// TIA Portal project "Asansör" (V16)

(* hardware
DEVICE "HMI_1"  TP900 Comfort
   slot 0: "HMI_1"  TP900 Comfort  6AV2 124-0JC01-0AX0  16.0.0.0
   slot 1: "HMI_RT_1"  TP900 Comfort  6AV2 124-0JC01-0AX0  16.0.0.0
   slot 5: "HMI_1.IE_CP_1"  PROFINET Interface  16.0.0.0
      slot 1: "PROFINET Interface_1"  PROFINET Interface
         slot 1: "Port_1"  Port
         slot 2: "Port_2"  Port
   slot 7: "HMI_1.MPI/DP_CP_1"  MPI/DP Interface  16.0.0.0
DEVICE "S71500/ET200MP station_1"  S7-1500 station
   slot 0: "Rail_0"  Rack  6ES7 590-1***0-0AA0
   slot 1: "PLC_1"  CPU 1513-1 PN  6ES7 513-1AL00-0AB0  V1.8
      slot 3: "CPU display_1"  6ES7591-1AA00-0AA0
      slot 32768: "PROFINET interface_1"  X1
         slot 32769: "Port_1"  X1 P1
         slot 32770: "Port_2"  X1 P2
*)

// ===== PLC "PLC_1"  CPU 1513-1 PN =====

VAR_GLOBAL   // PLC tag table "Default tag table"
   "Start" AT %M0.0 : Bool;
   "Start-System" AT %M0.1 : Bool;
   "P_TRIG" AT %M5.0 : Bool;
   "Stop" AT %M0.2 : Bool;
   "Low_Sensor" AT %M0.3 : Bool;
   "High_Sensor" AT %M0.4 : Bool;
   "P_TRIG1" AT %M5.1 : Bool;
   "Floor 1 button" AT %M0.5 : Bool;
   "P_TRIG2" AT %M5.2 : Bool;
   "Floor 1_Memory" AT %M0.6 : Bool;
   "Floor1_Sensor" AT %M0.7 : Bool;
   "P_TRIG3" AT %M5.3 : Bool;
   "Floor 2 button" AT %M1.0 : Bool;
   "P_TRIG4" AT %M5.4 : Bool;
   "Floor 2_Memory" AT %M1.1 : Bool;
   "Floor2_Sensor" AT %M1.2 : Bool;
   "P_TRIG5" AT %M5.5 : Bool;
   "Floor 3 button" AT %M1.3 : Bool;
   "Floor 3_Memory" AT %M1.4 : Bool;
   "P_TRIG6" AT %M5.6 : Bool;
   "Floor3_Sensor" AT %M1.5 : Bool;
   "P_TRIG7" AT %M5.7 : Bool;
   "P_TRIG8" AT %M6.1 : Bool;
   "Motor_Memory" AT %M1.6 : Bool;
   "Motor_Up" AT %M1.7 : Bool;
   "P_TRIG9" AT %M6.2 : Bool;
   "Memory2" AT %M2.0 : Bool;
   "Memory3" AT %M2.1 : Bool;
   "P_TRIG10" AT %M6.3 : Bool;
   "Motor_asagımemory" AT %M2.2 : Bool;
   "Motor_Down" AT %M2.3 : Bool;
   "P_TRIG11" AT %M6.4 : Bool;
   "Memory4" AT %M2.4 : Bool;
   "Memory5" AT %M2.5 : Bool;
END_VAR

DATA_BLOCK "Elevator"   // DB1
{ S7_Optimized_Access := 'TRUE' }
VERSION : 0.1
   VAR
      "Start System" : Bool;
      "Start--Stop" : Bool;
      "0_Floor" : Bool;
      "1_Floor" : Bool;
      "2_Floor" : Bool;
      Fan : Bool;
      Low_Sensor : Bool;
      High_Sensor : Bool;
      "1_Floor_Button" : Bool;
      "1_Floor_Sensor" : Bool;
      "2_Floor_Button" : Bool;
      "2_Floor_Sensor" : Bool;
      "3_Floor_Button" : Bool;
      "3_Floor_Sensor" : Bool;
      Motor_Up : Bool;
   END_VAR
BEGIN
END_DATA_BLOCK

ORGANIZATION_BLOCK "Main"   // OB1, LAD, ProgramCycle
TITLE = "Main Program Sweep (Cycle)"
{ S7_Optimized_Access := 'TRUE' }
VERSION : 0.1
   VAR_INPUT
      Initial_Call : Bool;   // Initial call of this OB
      Remanence : Bool;   // =True, if remanent data are available
   END_VAR
   VAR_TEMP   // added for the SCL form of the ladder/FBD networks
      _w1 : Bool;
      _w2 : Bool;
      _w3 : Bool;
      _w4 : Bool;
      _w5 : Bool;
      _w6 : Bool;
   END_VAR
BEGIN

REGION Network 1
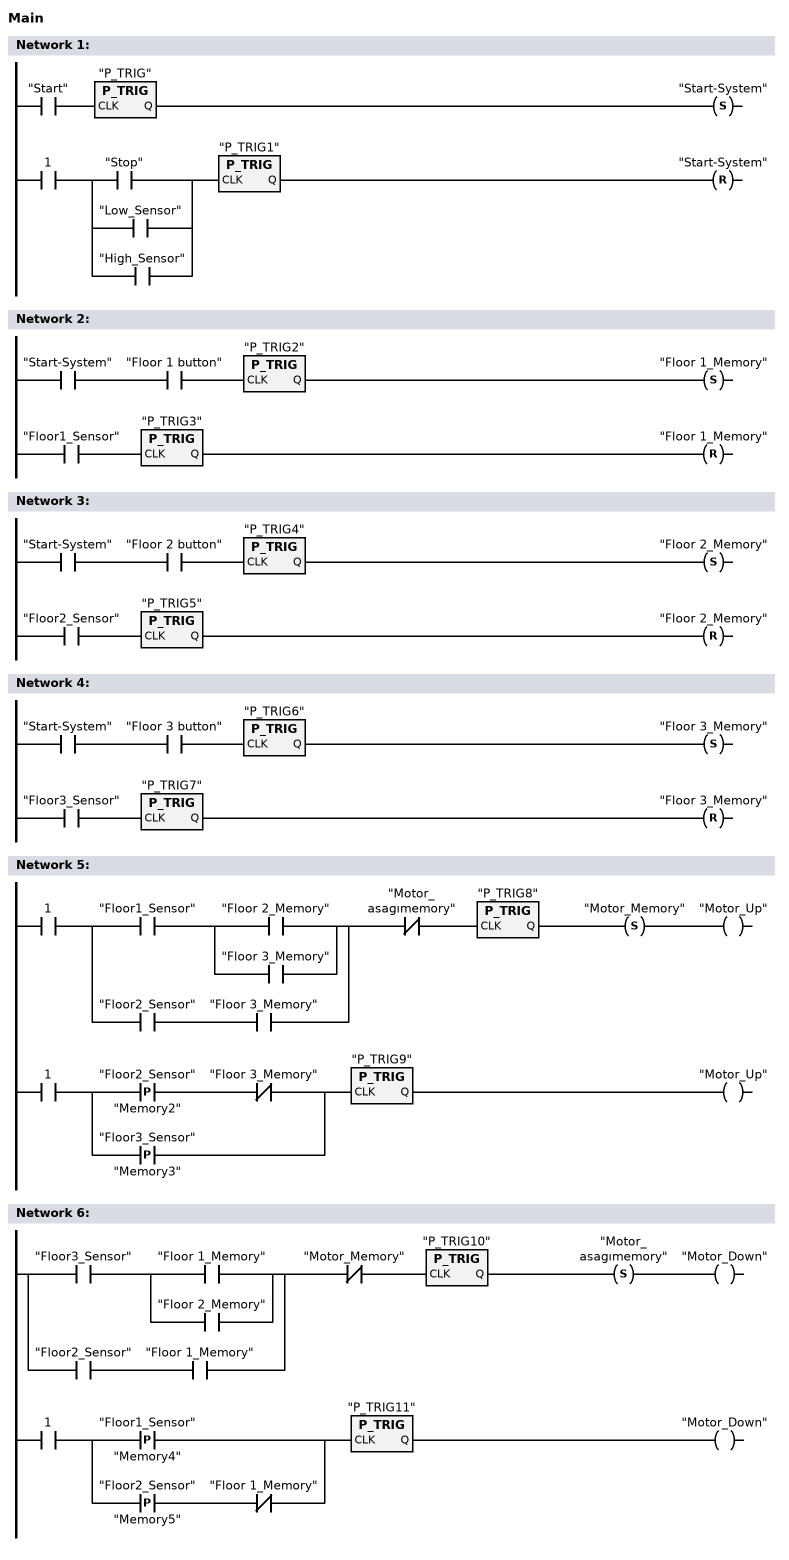
   RUNG wire#powerrail
      Contact( "Start" )
      P_Trig( "P_TRIG" )
      S_Coil( "Start-System" )
   END_RUNG
   RUNG wire#powerrail
      Contact( 1 )
      wire#w1
      Contact( "Stop" )
      wire#w2
      P_Trig( "P_TRIG1" )
      R_Coil( "Start-System" )
   END_RUNG
   RUNG wire#w1
      Contact( "Low_Sensor" )
   END_RUNG wire#w2
   RUNG wire#w1
      Contact( "High_Sensor" )
   END_RUNG wire#w2
   // the same network as SCL:
   #_w1 := "Start" AND NOT "P_TRIG";   // rising edge
   "P_TRIG" := "Start";
   IF #_w1 THEN "Start-System" := TRUE; END_IF;
   #_w2 := 1 AND ("Stop" OR "Low_Sensor" OR "High_Sensor");
   #_w3 := #_w2 AND NOT "P_TRIG1";   // rising edge
   "P_TRIG1" := #_w2;
   IF #_w3 THEN "Start-System" := FALSE; END_IF;
END_REGION

REGION Network 2
   RUNG wire#powerrail
      Contact( "Start-System" )
      Contact( "Floor 1 button" )
      P_Trig( "P_TRIG2" )
      S_Coil( "Floor 1_Memory" )
   END_RUNG
   RUNG wire#powerrail
      Contact( "Floor1_Sensor" )
      P_Trig( "P_TRIG3" )
      R_Coil( "Floor 1_Memory" )
   END_RUNG
   // the same network as SCL:
   #_w1 := "Start-System" AND "Floor 1 button";
   #_w2 := #_w1 AND NOT "P_TRIG2";   // rising edge
   "P_TRIG2" := #_w1;
   IF #_w2 THEN "Floor 1_Memory" := TRUE; END_IF;
   #_w3 := "Floor1_Sensor" AND NOT "P_TRIG3";   // rising edge
   "P_TRIG3" := "Floor1_Sensor";
   IF #_w3 THEN "Floor 1_Memory" := FALSE; END_IF;
END_REGION

REGION Network 3
   RUNG wire#powerrail
      Contact( "Start-System" )
      Contact( "Floor 2 button" )
      P_Trig( "P_TRIG4" )
      S_Coil( "Floor 2_Memory" )
   END_RUNG
   RUNG wire#powerrail
      Contact( "Floor2_Sensor" )
      P_Trig( "P_TRIG5" )
      R_Coil( "Floor 2_Memory" )
   END_RUNG
   // the same network as SCL:
   #_w1 := "Start-System" AND "Floor 2 button";
   #_w2 := #_w1 AND NOT "P_TRIG4";   // rising edge
   "P_TRIG4" := #_w1;
   IF #_w2 THEN "Floor 2_Memory" := TRUE; END_IF;
   #_w3 := "Floor2_Sensor" AND NOT "P_TRIG5";   // rising edge
   "P_TRIG5" := "Floor2_Sensor";
   IF #_w3 THEN "Floor 2_Memory" := FALSE; END_IF;
END_REGION

REGION Network 4
   RUNG wire#powerrail
      Contact( "Start-System" )
      Contact( "Floor 3 button" )
      P_Trig( "P_TRIG6" )
      S_Coil( "Floor 3_Memory" )
   END_RUNG
   RUNG wire#powerrail
      Contact( "Floor3_Sensor" )
      P_Trig( "P_TRIG7" )
      R_Coil( "Floor 3_Memory" )
   END_RUNG
   // the same network as SCL:
   #_w1 := "Start-System" AND "Floor 3 button";
   #_w2 := #_w1 AND NOT "P_TRIG6";   // rising edge
   "P_TRIG6" := #_w1;
   IF #_w2 THEN "Floor 3_Memory" := TRUE; END_IF;
   #_w3 := "Floor3_Sensor" AND NOT "P_TRIG7";   // rising edge
   "P_TRIG7" := "Floor3_Sensor";
   IF #_w3 THEN "Floor 3_Memory" := FALSE; END_IF;
END_REGION

REGION Network 5
   RUNG wire#powerrail
      Contact( 1 )
      wire#w1
      Contact( "Floor1_Sensor" )
      wire#w2
      Contact( "Floor 2_Memory" )
      wire#w3
      I_Contact( "Motor_asagımemory" )
      P_Trig( "P_TRIG8" )
      S_Coil( "Motor_Memory" )
      Coil( "Motor_Up" )
   END_RUNG
   RUNG wire#w2
      Contact( "Floor 3_Memory" )
   END_RUNG wire#w3
   RUNG wire#w1
      Contact( "Floor2_Sensor" )
      Contact( "Floor 3_Memory" )
   END_RUNG wire#w3
   RUNG wire#powerrail
      Contact( 1 )
      wire#w4
      P_Contact(operand := "Floor2_Sensor", bit := "Memory2")
      I_Contact( "Floor 3_Memory" )
      wire#w5
      P_Trig( "P_TRIG9" )
      Coil( "Motor_Up" )
   END_RUNG
   RUNG wire#w4
      P_Contact(operand := "Floor3_Sensor", bit := "Memory3")
   END_RUNG wire#w5
   // the same network as SCL:
   #_w1 := 1 AND (("Floor1_Sensor" AND ("Floor 2_Memory" OR "Floor 3_Memory")) OR ("Floor2_Sensor" AND "Floor 3_Memory")) AND NOT "Motor_asagımemory";
   #_w2 := #_w1 AND NOT "P_TRIG8";   // rising edge
   "P_TRIG8" := #_w1;
   IF #_w2 THEN "Motor_Memory" := TRUE; END_IF;
   "Motor_Up" := #_w2;
   #_w3 := 1 AND "Floor2_Sensor" AND NOT "Memory2";   // rising edge of "Floor2_Sensor"
   "Memory2" := "Floor2_Sensor";
   #_w4 := 1 AND "Floor3_Sensor" AND NOT "Memory3";   // rising edge of "Floor3_Sensor"
   "Memory3" := "Floor3_Sensor";
   #_w5 := (#_w3 AND NOT "Floor 3_Memory") OR #_w4;
   #_w6 := #_w5 AND NOT "P_TRIG9";   // rising edge
   "P_TRIG9" := #_w5;
   "Motor_Up" := #_w6;
END_REGION

REGION Network 6
   RUNG wire#powerrail
      Contact( "Floor3_Sensor" )
      wire#w1
      Contact( "Floor 1_Memory" )
      wire#w2
      I_Contact( "Motor_Memory" )
      P_Trig( "P_TRIG10" )
      S_Coil( "Motor_asagımemory" )
      Coil( "Motor_Down" )
   END_RUNG
   RUNG wire#w1
      Contact( "Floor 2_Memory" )
   END_RUNG wire#w2
   RUNG wire#powerrail
      Contact( "Floor2_Sensor" )
      Contact( "Floor 1_Memory" )
   END_RUNG wire#w2
   RUNG wire#powerrail
      Contact( 1 )
      wire#w3
      P_Contact(operand := "Floor1_Sensor", bit := "Memory4")
      wire#w4
      P_Trig( "P_TRIG11" )
      Coil( "Motor_Down" )
   END_RUNG
   RUNG wire#w3
      P_Contact(operand := "Floor2_Sensor", bit := "Memory5")
      I_Contact( "Floor 1_Memory" )
   END_RUNG wire#w4
   // the same network as SCL:
   #_w1 := (("Floor3_Sensor" AND ("Floor 1_Memory" OR "Floor 2_Memory")) OR ("Floor2_Sensor" AND "Floor 1_Memory")) AND NOT "Motor_Memory";
   #_w2 := #_w1 AND NOT "P_TRIG10";   // rising edge
   "P_TRIG10" := #_w1;
   IF #_w2 THEN "Motor_asagımemory" := TRUE; END_IF;
   "Motor_Down" := #_w2;
   #_w3 := 1 AND "Floor1_Sensor" AND NOT "Memory4";   // rising edge of "Floor1_Sensor"
   "Memory4" := "Floor1_Sensor";
   #_w4 := 1 AND "Floor2_Sensor" AND NOT "Memory5";   // rising edge of "Floor2_Sensor"
   "Memory5" := "Floor2_Sensor";
   #_w5 := #_w3 OR (#_w4 AND NOT "Floor 1_Memory");
   #_w6 := #_w5 AND NOT "P_TRIG11";   // rising edge
   "P_TRIG11" := #_w5;
   "Motor_Down" := #_w6;
END_REGION
END_ORGANIZATION_BLOCK

(* ===== HMI "HMI_RT_1" =====
system functions are stored by id; their names below are inferred from use
connection "HMI_Connection_1": ETHERNET, S7_1500_OMS

HMI tags "Default tag table"
   "Tag_ScreenNumber" : UInt, internal
   "Fan" : Bool = PLC Fan AT %M0.0, 1 s
   "Button for 1 floor" : Bool = PLC "Button for 1 floor" AT %M0.7, 1 s
   "Button for 2 floor" : Bool = PLC "Button for 2 floor" AT %M0.6, 1 s
   "Start the motor upwards" : Bool = PLC "Start the motor upwards" AT %M0.3, 1 s

screen "Root screen" 800x420, template "Template_1"
   on GenerateScreen: SetTag("Tag_ScreenNumber", 1)
   Button "Button_4" at 11,32 size 99x32; TextOff 'Fan Start-Stop'
      on Press: function_b14e0dd5("Fan", 0)
   Circle "Circle_4" at 158,27 size 48x48
      Appearance <- "Fan"
   Button "Button_1" at 11,85 size 170x32; TextOff 'Button for 1 floor inside'
      on Press: InvertBit("Button for 1 floor")
   Button "Button_2" at 11,142 size 170x32; TextOff 'Button for 2 floor inside'
      on Press: InvertBit("Button for 2 floor")
   Circle "Circle_1" at 213,74 size 48x48
      Appearance <- "Button for 1 floor"
   Circle "Circle_2" at 214,132 size 48x48
      Appearance <- "Button for 2 floor"
   TextField "Text field_1" at 382,26 size 161x20; Text 'Start Motor upwards'
   Circle "Circle_3" at 550,13 size 48x48
      Appearance <- "Start the motor upwards"

Template "Template_1" 800x420
   Button "Exit" at 720,360 size 78x58; TextOff 'Exit'; PictureOff "ExitRuntime_TP900_Comfort_TR"; PictureOn "ExitRuntime_TP900_Comfort_TR"
      on Release: StopRuntime(0)
   Button "Template_Button" at 640,360 size 78x58; TextOff 'Text'
   Button "Template_Button_1" at 560,360 size 78x58; TextOff 'Text'
   Button "Template_Button_2" at 480,360 size 78x58; TextOff 'Text'
   Button "Template_Button_3" at 400,360 size 78x58; TextOff 'Text'
   Button "Template_Button_4" at 321,360 size 78x58; TextOff 'Text'
   Button "Template_Button_5" at 241,360 size 78x58; TextOff 'Text'
   Button "Template_Button_6" at 161,360 size 78x58; TextOff 'Text'
   Button "Alarms" at 81,360 size 78x58; TextOff 'Alarms'; PictureOff "AlarmDisplay_TP900_Comfort_TR"; PictureOn "AlarmDisplay_TP900_Comfort_TR"
      on Release: function_ef3f5d25("Alarm window_Unacknowledged", -1)
   Button "Start screen" at 1,360 size 78x58; TextOff 'Start screen'; PictureOff "NavigateHome_TP900_Comfort_TR"; PictureOn "NavigateHome_TP900_Comfort_TR"
      on Release: ActivateScreen("Root screen", 0)
*)